SYSTEM StopperingModule (* Module Stoppering, generated from its module specification *)
  (* Standard: 61499-2 *)
  APPLICATION Stoppering (* Module Stoppering on target pc (localhost, IO modbus; generated by modgen) *)
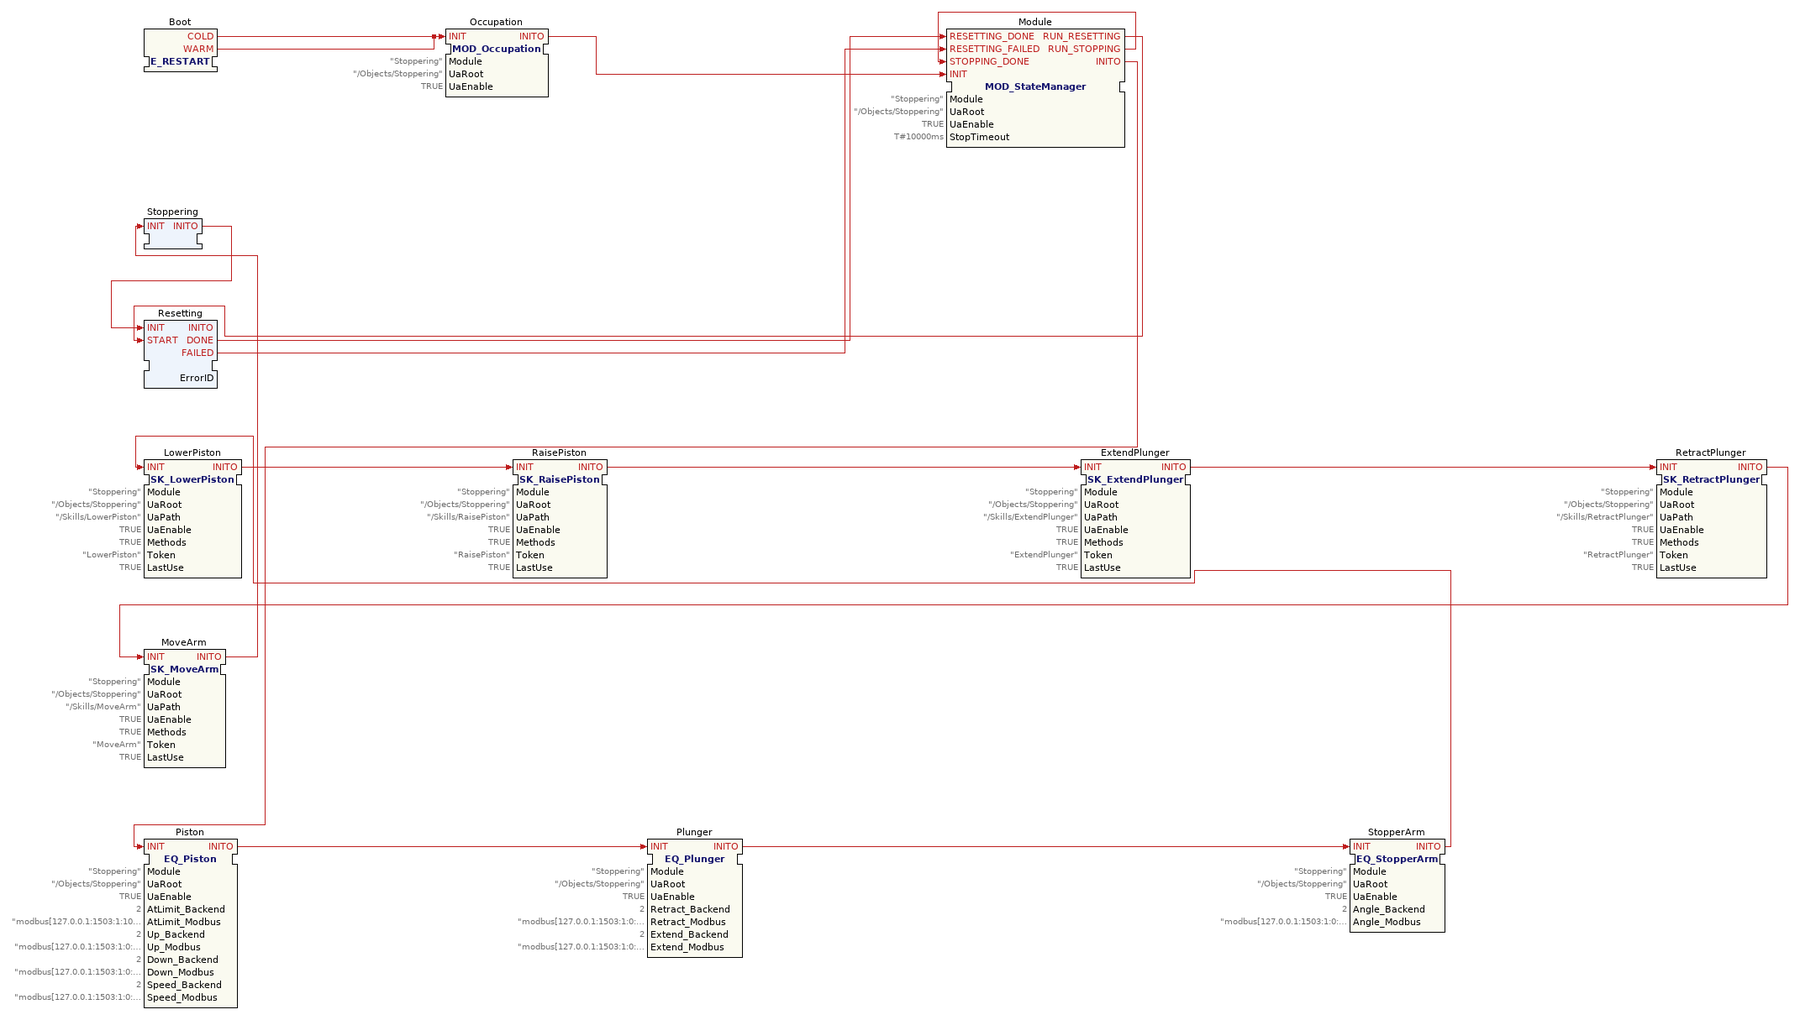
    (* Group ModuleLevel: Module level: occupation, PackML state manager, start-up and the target's IO lines *)
    (* Group ModuleLevelSkills: Module level skills: Control + Execute (+ Stop) sequences of skill primitives; OPC UA /Skills/<name> *)
    (* Group Procedures: Procedures the module state manager runs while Resetting and Stopping *)
    (* Group SkillPrimitives: Skill primitives: one equipment command until a sensor or a time; OPC UA /Skills/<name> *)
    (* Group EquipmentIO: Equipment IO: the only owners of the IO points; skills command them over local channels *)
    FBS
      Boot : iec61499::events::E_RESTART; {SET_ATTRIBUTE(GroupName, ModuleLevel)}
      Occupation : modlib::MOD_Occupation(Module := "Stoppering", UaRoot := "/Objects/Stoppering", UaEnable := TRUE); {SET_ATTRIBUTE(GroupName, ModuleLevel)}
      Module : modlib::MOD_StateManager(Module := "Stoppering", UaRoot := "/Objects/Stoppering", UaEnable := TRUE, StopTimeout := T#10000ms); {SET_ATTRIBUTE(GroupName, ModuleLevel)}
      Piston : stoppering::EQ_Piston(Module := "Stoppering", UaRoot := "/Objects/Stoppering", UaEnable := TRUE, AtLimit_Backend := 2, AtLimit_Modbus := "modbus[127.0.0.1:1503:1:10:d0:]", Up_Backend := 2, Up_Modbus := "modbus[127.0.0.1:1503:1:0::c0]", Down_Backend := 2, Down_Modbus := "modbus[127.0.0.1:1503:1:0::c1]", Speed_Backend := 2, Speed_Modbus := "modbus[127.0.0.1:1503:1:0::h0]"); {SET_ATTRIBUTE(GroupName, EquipmentIO)}
      Plunger : stoppering::EQ_Plunger(Module := "Stoppering", UaRoot := "/Objects/Stoppering", UaEnable := TRUE, Retract_Backend := 2, Retract_Modbus := "modbus[127.0.0.1:1503:1:0::c2]", Extend_Backend := 2, Extend_Modbus := "modbus[127.0.0.1:1503:1:0::c3]"); {SET_ATTRIBUTE(GroupName, EquipmentIO)}
      StopperArm : stoppering::EQ_StopperArm(Module := "Stoppering", UaRoot := "/Objects/Stoppering", UaEnable := TRUE, Angle_Backend := 2, Angle_Modbus := "modbus[127.0.0.1:1503:1:0::h1]"); {SET_ATTRIBUTE(GroupName, EquipmentIO)}
      LowerPiston : stoppering::SK_LowerPiston(Module := "Stoppering", UaRoot := "/Objects/Stoppering", UaPath := "/Skills/LowerPiston", UaEnable := TRUE, Methods := TRUE, Token := "LowerPiston", LastUse := TRUE); {SET_ATTRIBUTE(GroupName, SkillPrimitives)}
      RaisePiston : stoppering::SK_RaisePiston(Module := "Stoppering", UaRoot := "/Objects/Stoppering", UaPath := "/Skills/RaisePiston", UaEnable := TRUE, Methods := TRUE, Token := "RaisePiston", LastUse := TRUE); {SET_ATTRIBUTE(GroupName, SkillPrimitives)}
      ExtendPlunger : stoppering::SK_ExtendPlunger(Module := "Stoppering", UaRoot := "/Objects/Stoppering", UaPath := "/Skills/ExtendPlunger", UaEnable := TRUE, Methods := TRUE, Token := "ExtendPlunger", LastUse := TRUE); {SET_ATTRIBUTE(GroupName, SkillPrimitives)}
      RetractPlunger : stoppering::SK_RetractPlunger(Module := "Stoppering", UaRoot := "/Objects/Stoppering", UaPath := "/Skills/RetractPlunger", UaEnable := TRUE, Methods := TRUE, Token := "RetractPlunger", LastUse := TRUE); {SET_ATTRIBUTE(GroupName, SkillPrimitives)}
      MoveArm : stoppering::SK_MoveArm(Module := "Stoppering", UaRoot := "/Objects/Stoppering", UaPath := "/Skills/MoveArm", UaEnable := TRUE, Methods := TRUE, Token := "MoveArm", LastUse := TRUE); {SET_ATTRIBUTE(GroupName, SkillPrimitives)}
    END_FBS
    SUBAPPLICATION Stoppering (* Module level skill Stoppering: Piston to the working position, place the stopper with the servo, plunge, piston up (runStopperingCycle) *)
      {SET_ATTRIBUTE(GroupName, ModuleLevelSkills)}
      EVENT_INPUT
        INIT : EInit;
      END_EVENT
      EVENT_OUTPUT
        INITO : EInit;
      END_EVENT
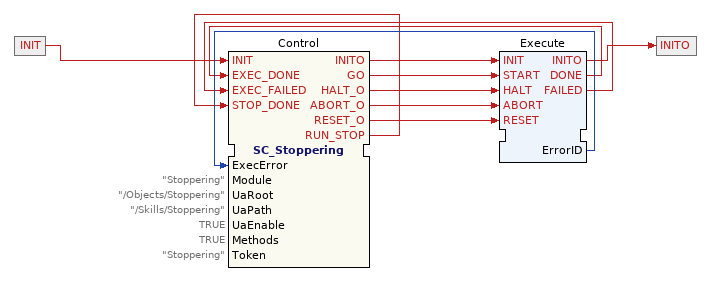
      FBS
        Control : stoppering::SC_Stoppering(Module := "Stoppering", UaRoot := "/Objects/Stoppering", UaPath := "/Skills/Stoppering", UaEnable := TRUE, Methods := TRUE, Token := "Stoppering");
      END_FBS
      SUBAPPLICATION Execute (* Stoppering: execute sequence *)
        EVENT_INPUT
          INIT : EInit;
          START;
          HALT;
          ABORT;
          RESET;
        END_EVENT
        EVENT_OUTPUT
          INITO : EInit;
          DONE;
          FAILED WITH ErrorID;
        END_EVENT
        VAR_OUTPUT
          ErrorID : UINT;
        END_VAR
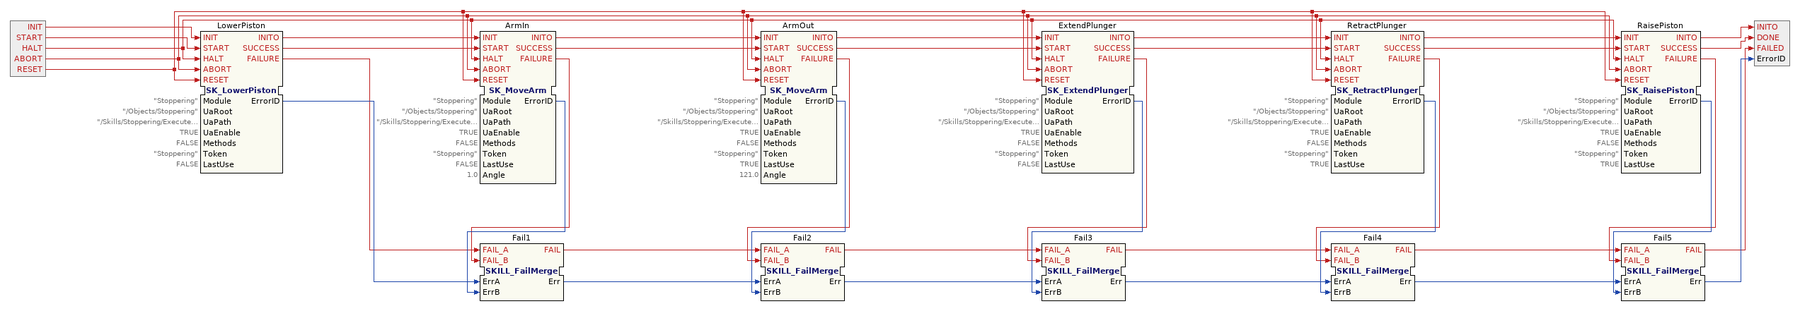
        FBS
          LowerPiston : stoppering::SK_LowerPiston(Module := "Stoppering", UaRoot := "/Objects/Stoppering", UaPath := "/Skills/Stoppering/Execute/LowerPiston", UaEnable := TRUE, Methods := FALSE, Token := "Stoppering", LastUse := FALSE);
          ArmIn : stoppering::SK_MoveArm(Module := "Stoppering", UaRoot := "/Objects/Stoppering", UaPath := "/Skills/Stoppering/Execute/ArmIn", UaEnable := TRUE, Methods := FALSE, Token := "Stoppering", LastUse := FALSE, Angle := 1.0);
          ArmOut : stoppering::SK_MoveArm(Module := "Stoppering", UaRoot := "/Objects/Stoppering", UaPath := "/Skills/Stoppering/Execute/ArmOut", UaEnable := TRUE, Methods := FALSE, Token := "Stoppering", LastUse := TRUE, Angle := 121.0);
          ExtendPlunger : stoppering::SK_ExtendPlunger(Module := "Stoppering", UaRoot := "/Objects/Stoppering", UaPath := "/Skills/Stoppering/Execute/ExtendPlunger", UaEnable := TRUE, Methods := FALSE, Token := "Stoppering", LastUse := FALSE);
          RetractPlunger : stoppering::SK_RetractPlunger(Module := "Stoppering", UaRoot := "/Objects/Stoppering", UaPath := "/Skills/Stoppering/Execute/RetractPlunger", UaEnable := TRUE, Methods := FALSE, Token := "Stoppering", LastUse := TRUE);
          RaisePiston : stoppering::SK_RaisePiston(Module := "Stoppering", UaRoot := "/Objects/Stoppering", UaPath := "/Skills/Stoppering/Execute/RaisePiston", UaEnable := TRUE, Methods := FALSE, Token := "Stoppering", LastUse := TRUE);
          Fail1 : modlib::SKILL_FailMerge;
          Fail2 : modlib::SKILL_FailMerge;
          Fail3 : modlib::SKILL_FailMerge;
          Fail4 : modlib::SKILL_FailMerge;
          Fail5 : modlib::SKILL_FailMerge;
        END_FBS
        EVENT_CONNECTIONS
          INIT TO LowerPiston.INIT;
          RaisePiston.INITO TO INITO;
          START TO LowerPiston.START;
          RaisePiston.SUCCESS TO DONE;
          LowerPiston.INITO TO ArmIn.INIT;
          LowerPiston.SUCCESS TO ArmIn.START;
          ArmIn.INITO TO ArmOut.INIT;
          ArmIn.SUCCESS TO ArmOut.START;
          ArmOut.INITO TO ExtendPlunger.INIT;
          ArmOut.SUCCESS TO ExtendPlunger.START;
          ExtendPlunger.INITO TO RetractPlunger.INIT;
          ExtendPlunger.SUCCESS TO RetractPlunger.START;
          RetractPlunger.INITO TO RaisePiston.INIT;
          RetractPlunger.SUCCESS TO RaisePiston.START;
          HALT TO LowerPiston.HALT;
          HALT TO ArmIn.HALT;
          HALT TO ArmOut.HALT;
          HALT TO ExtendPlunger.HALT;
          HALT TO RetractPlunger.HALT;
          HALT TO RaisePiston.HALT;
          ABORT TO LowerPiston.ABORT;
          ABORT TO ArmIn.ABORT;
          ABORT TO ArmOut.ABORT;
          ABORT TO ExtendPlunger.ABORT;
          ABORT TO RetractPlunger.ABORT;
          ABORT TO RaisePiston.ABORT;
          RESET TO LowerPiston.RESET;
          RESET TO ArmIn.RESET;
          RESET TO ArmOut.RESET;
          RESET TO ExtendPlunger.RESET;
          RESET TO RetractPlunger.RESET;
          RESET TO RaisePiston.RESET;
          LowerPiston.FAILURE TO Fail1.FAIL_A;
          ArmIn.FAILURE TO Fail1.FAIL_B;
          Fail1.FAIL TO Fail2.FAIL_A;
          ArmOut.FAILURE TO Fail2.FAIL_B;
          Fail2.FAIL TO Fail3.FAIL_A;
          ExtendPlunger.FAILURE TO Fail3.FAIL_B;
          Fail3.FAIL TO Fail4.FAIL_A;
          RetractPlunger.FAILURE TO Fail4.FAIL_B;
          Fail4.FAIL TO Fail5.FAIL_A;
          RaisePiston.FAILURE TO Fail5.FAIL_B;
          Fail5.FAIL TO FAILED;
        END_CONNECTIONS
        DATA_CONNECTIONS
          LowerPiston.ErrorID TO Fail1.ErrA;
          ArmIn.ErrorID TO Fail1.ErrB;
          Fail1.Err TO Fail2.ErrA;
          ArmOut.ErrorID TO Fail2.ErrB;
          Fail2.Err TO Fail3.ErrA;
          ExtendPlunger.ErrorID TO Fail3.ErrB;
          Fail3.Err TO Fail4.ErrA;
          RetractPlunger.ErrorID TO Fail4.ErrB;
          Fail4.Err TO Fail5.ErrA;
          RaisePiston.ErrorID TO Fail5.ErrB;
          Fail5.Err TO ErrorID;
        END_CONNECTIONS
      END_SUBAPPLICATION
      EVENT_CONNECTIONS
        INIT TO Control.INIT;
        Control.INITO TO Execute.INIT;
        Control.GO TO Execute.START;
        Control.HALT_O TO Execute.HALT;
        Control.ABORT_O TO Execute.ABORT;
        Control.RESET_O TO Execute.RESET;
        Execute.DONE TO Control.EXEC_DONE;
        Execute.FAILED TO Control.EXEC_FAILED;
        Execute.INITO TO INITO;
        Control.RUN_STOP TO Control.STOP_DONE;
      END_CONNECTIONS
      DATA_CONNECTIONS
        Execute.ErrorID TO Control.ExecError;
      END_CONNECTIONS
    END_SUBAPPLICATION
    SUBAPPLICATION Resetting (* Procedure the module runs while Resetting *)
      {SET_ATTRIBUTE(GroupName, Procedures)}
      EVENT_INPUT
        INIT : EInit;
        START;
      END_EVENT
      EVENT_OUTPUT
        INITO : EInit;
        DONE;
        FAILED WITH ErrorID;
      END_EVENT
      VAR_OUTPUT
        ErrorID : UINT;
      END_VAR
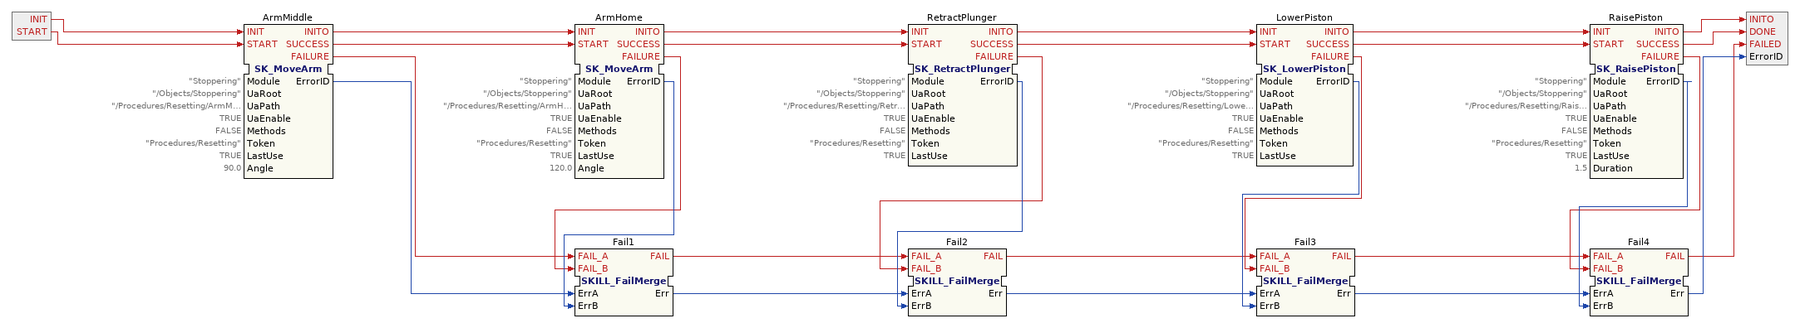
      FBS
        ArmMiddle : stoppering::SK_MoveArm(Module := "Stoppering", UaRoot := "/Objects/Stoppering", UaPath := "/Procedures/Resetting/ArmMiddle", UaEnable := TRUE, Methods := FALSE, Token := "Procedures/Resetting", LastUse := TRUE, Angle := 90.0);
        ArmHome : stoppering::SK_MoveArm(Module := "Stoppering", UaRoot := "/Objects/Stoppering", UaPath := "/Procedures/Resetting/ArmHome", UaEnable := TRUE, Methods := FALSE, Token := "Procedures/Resetting", LastUse := TRUE, Angle := 120.0);
        RetractPlunger : stoppering::SK_RetractPlunger(Module := "Stoppering", UaRoot := "/Objects/Stoppering", UaPath := "/Procedures/Resetting/RetractPlunger", UaEnable := TRUE, Methods := FALSE, Token := "Procedures/Resetting", LastUse := TRUE);
        LowerPiston : stoppering::SK_LowerPiston(Module := "Stoppering", UaRoot := "/Objects/Stoppering", UaPath := "/Procedures/Resetting/LowerPiston", UaEnable := TRUE, Methods := FALSE, Token := "Procedures/Resetting", LastUse := TRUE);
        RaisePiston : stoppering::SK_RaisePiston(Module := "Stoppering", UaRoot := "/Objects/Stoppering", UaPath := "/Procedures/Resetting/RaisePiston", UaEnable := TRUE, Methods := FALSE, Token := "Procedures/Resetting", LastUse := TRUE, Duration := 1.5);
        Fail1 : modlib::SKILL_FailMerge;
        Fail2 : modlib::SKILL_FailMerge;
        Fail3 : modlib::SKILL_FailMerge;
        Fail4 : modlib::SKILL_FailMerge;
      END_FBS
      EVENT_CONNECTIONS
        INIT TO ArmMiddle.INIT;
        RaisePiston.INITO TO INITO;
        START TO ArmMiddle.START;
        RaisePiston.SUCCESS TO DONE;
        ArmMiddle.INITO TO ArmHome.INIT;
        ArmMiddle.SUCCESS TO ArmHome.START;
        ArmHome.INITO TO RetractPlunger.INIT;
        ArmHome.SUCCESS TO RetractPlunger.START;
        RetractPlunger.INITO TO LowerPiston.INIT;
        RetractPlunger.SUCCESS TO LowerPiston.START;
        LowerPiston.INITO TO RaisePiston.INIT;
        LowerPiston.SUCCESS TO RaisePiston.START;
        ArmMiddle.FAILURE TO Fail1.FAIL_A;
        ArmHome.FAILURE TO Fail1.FAIL_B;
        Fail1.FAIL TO Fail2.FAIL_A;
        RetractPlunger.FAILURE TO Fail2.FAIL_B;
        Fail2.FAIL TO Fail3.FAIL_A;
        LowerPiston.FAILURE TO Fail3.FAIL_B;
        Fail3.FAIL TO Fail4.FAIL_A;
        RaisePiston.FAILURE TO Fail4.FAIL_B;
        Fail4.FAIL TO FAILED;
      END_CONNECTIONS
      DATA_CONNECTIONS
        ArmMiddle.ErrorID TO Fail1.ErrA;
        ArmHome.ErrorID TO Fail1.ErrB;
        Fail1.Err TO Fail2.ErrA;
        RetractPlunger.ErrorID TO Fail2.ErrB;
        Fail2.Err TO Fail3.ErrA;
        LowerPiston.ErrorID TO Fail3.ErrB;
        Fail3.Err TO Fail4.ErrA;
        RaisePiston.ErrorID TO Fail4.ErrB;
        Fail4.Err TO ErrorID;
      END_CONNECTIONS
    END_SUBAPPLICATION
    EVENT_CONNECTIONS
      Boot.COLD TO Occupation.INIT;
      Boot.WARM TO Occupation.INIT;
      Module.RUN_RESETTING TO Resetting.START;
      Resetting.DONE TO Module.RESETTING_DONE;
      Resetting.FAILED TO Module.RESETTING_FAILED;
      Module.RUN_STOPPING TO Module.STOPPING_DONE;
      Occupation.INITO TO Module.INIT;
      Module.INITO TO Piston.INIT;
      Piston.INITO TO Plunger.INIT;
      Plunger.INITO TO StopperArm.INIT;
      StopperArm.INITO TO LowerPiston.INIT;
      LowerPiston.INITO TO RaisePiston.INIT;
      RaisePiston.INITO TO ExtendPlunger.INIT;
      ExtendPlunger.INITO TO RetractPlunger.INIT;
      RetractPlunger.INITO TO MoveArm.INIT;
      MoveArm.INITO TO Stoppering.INIT;
      Stoppering.INITO TO Resetting.INIT;
    END_CONNECTIONS
  END_APPLICATION
  APPLICATION Stoppering_pi (* Module Stoppering on target pi (stoppering-pi, IO gpio; generated by modgen) *)
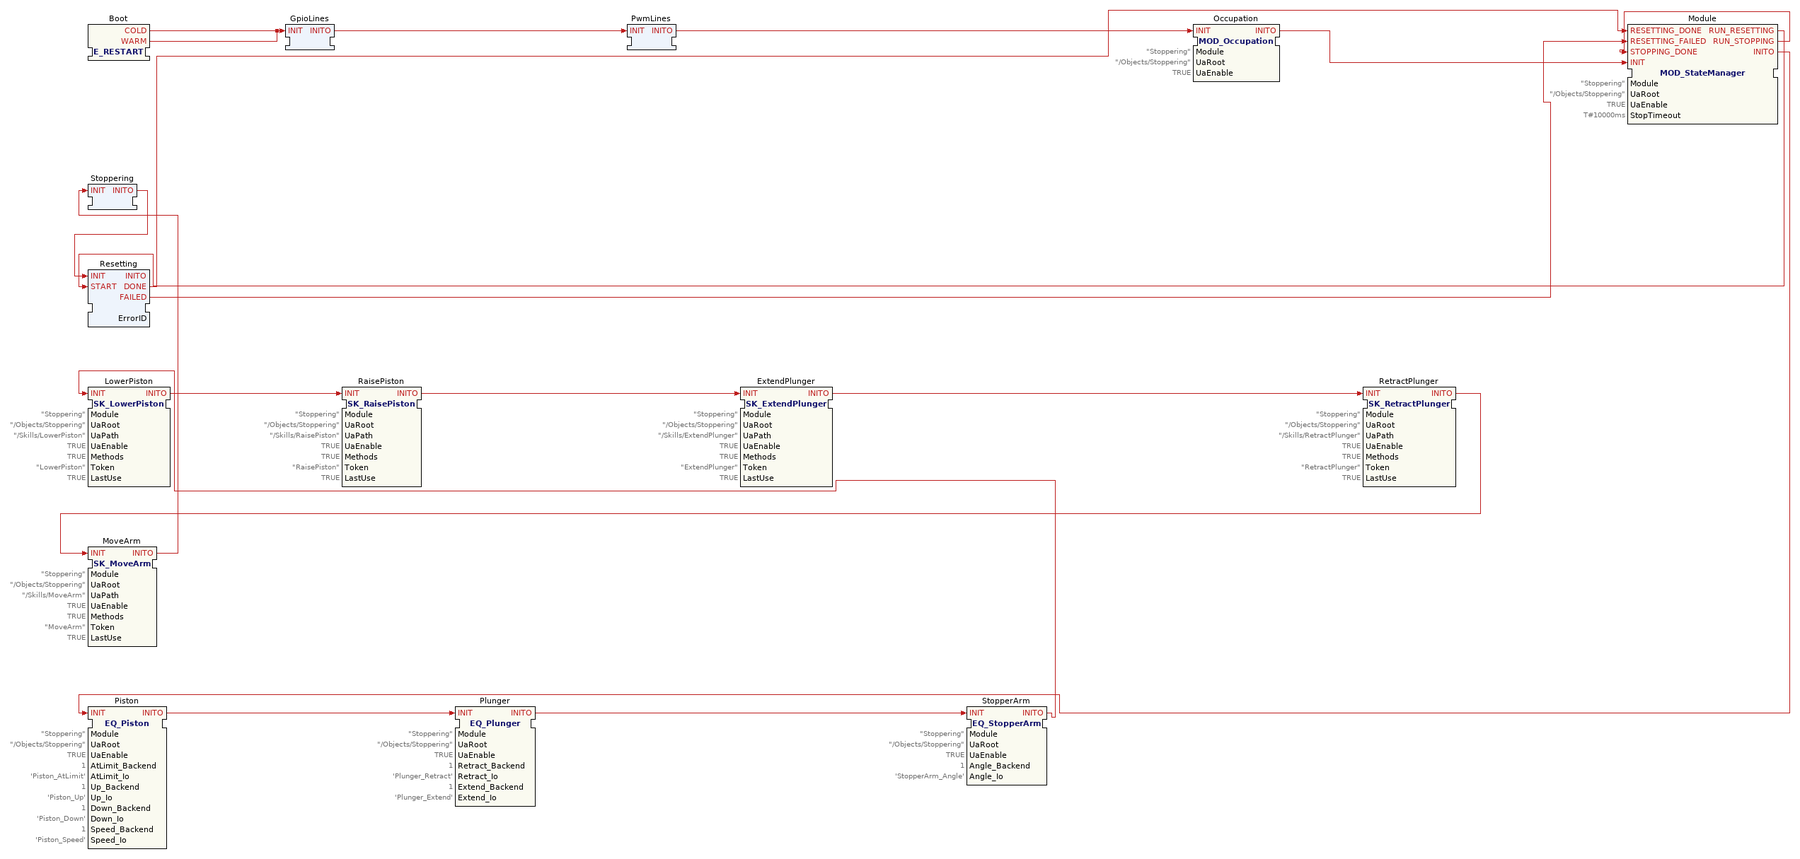
    (* Group ModuleLevel: Module level: occupation, PackML state manager, start-up and the target's IO lines *)
    (* Group ModuleLevelSkills: Module level skills: Control + Execute (+ Stop) sequences of skill primitives; OPC UA /Skills/<name> *)
    (* Group Procedures: Procedures the module state manager runs while Resetting and Stopping *)
    (* Group SkillPrimitives: Skill primitives: one equipment command until a sensor or a time; OPC UA /Skills/<name> *)
    (* Group EquipmentIO: Equipment IO: the only owners of the IO points; skills command them over local channels *)
    FBS
      Boot : iec61499::events::E_RESTART; {SET_ATTRIBUTE(GroupName, ModuleLevel)}
      Occupation : modlib::MOD_Occupation(Module := "Stoppering", UaRoot := "/Objects/Stoppering", UaEnable := TRUE); {SET_ATTRIBUTE(GroupName, ModuleLevel)}
      Module : modlib::MOD_StateManager(Module := "Stoppering", UaRoot := "/Objects/Stoppering", UaEnable := TRUE, StopTimeout := T#10000ms); {SET_ATTRIBUTE(GroupName, ModuleLevel)}
      Piston : stoppering::EQ_Piston(Module := "Stoppering", UaRoot := "/Objects/Stoppering", UaEnable := TRUE, AtLimit_Backend := 1, AtLimit_Io := 'Piston_AtLimit', Up_Backend := 1, Up_Io := 'Piston_Up', Down_Backend := 1, Down_Io := 'Piston_Down', Speed_Backend := 1, Speed_Io := 'Piston_Speed'); {SET_ATTRIBUTE(GroupName, EquipmentIO)}
      Plunger : stoppering::EQ_Plunger(Module := "Stoppering", UaRoot := "/Objects/Stoppering", UaEnable := TRUE, Retract_Backend := 1, Retract_Io := 'Plunger_Retract', Extend_Backend := 1, Extend_Io := 'Plunger_Extend'); {SET_ATTRIBUTE(GroupName, EquipmentIO)}
      StopperArm : stoppering::EQ_StopperArm(Module := "Stoppering", UaRoot := "/Objects/Stoppering", UaEnable := TRUE, Angle_Backend := 1, Angle_Io := 'StopperArm_Angle'); {SET_ATTRIBUTE(GroupName, EquipmentIO)}
      LowerPiston : stoppering::SK_LowerPiston(Module := "Stoppering", UaRoot := "/Objects/Stoppering", UaPath := "/Skills/LowerPiston", UaEnable := TRUE, Methods := TRUE, Token := "LowerPiston", LastUse := TRUE); {SET_ATTRIBUTE(GroupName, SkillPrimitives)}
      RaisePiston : stoppering::SK_RaisePiston(Module := "Stoppering", UaRoot := "/Objects/Stoppering", UaPath := "/Skills/RaisePiston", UaEnable := TRUE, Methods := TRUE, Token := "RaisePiston", LastUse := TRUE); {SET_ATTRIBUTE(GroupName, SkillPrimitives)}
      ExtendPlunger : stoppering::SK_ExtendPlunger(Module := "Stoppering", UaRoot := "/Objects/Stoppering", UaPath := "/Skills/ExtendPlunger", UaEnable := TRUE, Methods := TRUE, Token := "ExtendPlunger", LastUse := TRUE); {SET_ATTRIBUTE(GroupName, SkillPrimitives)}
      RetractPlunger : stoppering::SK_RetractPlunger(Module := "Stoppering", UaRoot := "/Objects/Stoppering", UaPath := "/Skills/RetractPlunger", UaEnable := TRUE, Methods := TRUE, Token := "RetractPlunger", LastUse := TRUE); {SET_ATTRIBUTE(GroupName, SkillPrimitives)}
      MoveArm : stoppering::SK_MoveArm(Module := "Stoppering", UaRoot := "/Objects/Stoppering", UaPath := "/Skills/MoveArm", UaEnable := TRUE, Methods := TRUE, Token := "MoveArm", LastUse := TRUE); {SET_ATTRIBUTE(GroupName, SkillPrimitives)}
    END_FBS
    SUBAPPLICATION GpioLines (* GPIO lines of the equipment's IO points (Linux /dev/gpiochip) *)
      {SET_ATTRIBUTE(GroupName, ModuleLevel)}
      EVENT_INPUT
        INIT : EInit;
      END_EVENT
      EVENT_OUTPUT
        INITO : EInit;
      END_EVENT
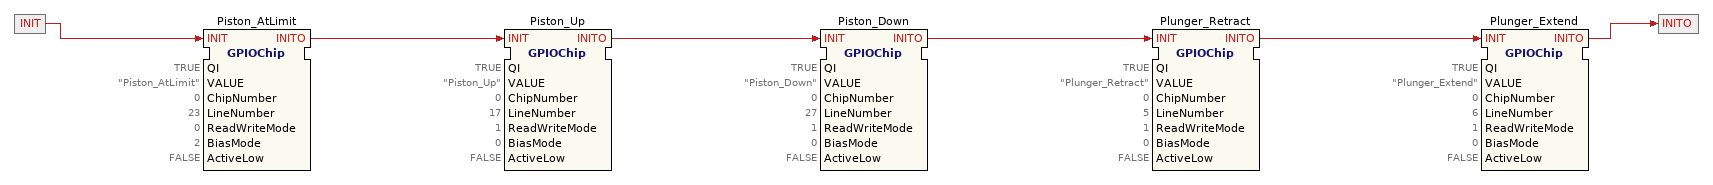
      FBS
        Piston_AtLimit : eclipse4diac::io::gpiochip::GPIOChip(QI := TRUE, VALUE := "Piston_AtLimit", ChipNumber := 0, LineNumber := 23, ReadWriteMode := 0, BiasMode := 2, ActiveLow := FALSE);
        Piston_Up : eclipse4diac::io::gpiochip::GPIOChip(QI := TRUE, VALUE := "Piston_Up", ChipNumber := 0, LineNumber := 17, ReadWriteMode := 1, BiasMode := 0, ActiveLow := FALSE);
        Piston_Down : eclipse4diac::io::gpiochip::GPIOChip(QI := TRUE, VALUE := "Piston_Down", ChipNumber := 0, LineNumber := 27, ReadWriteMode := 1, BiasMode := 0, ActiveLow := FALSE);
        Plunger_Retract : eclipse4diac::io::gpiochip::GPIOChip(QI := TRUE, VALUE := "Plunger_Retract", ChipNumber := 0, LineNumber := 5, ReadWriteMode := 1, BiasMode := 0, ActiveLow := FALSE);
        Plunger_Extend : eclipse4diac::io::gpiochip::GPIOChip(QI := TRUE, VALUE := "Plunger_Extend", ChipNumber := 0, LineNumber := 6, ReadWriteMode := 1, BiasMode := 0, ActiveLow := FALSE);
      END_FBS
      EVENT_CONNECTIONS
        INIT TO Piston_AtLimit.INIT;
        Plunger_Extend.INITO TO INITO;
        Piston_AtLimit.INITO TO Piston_Up.INIT;
        Piston_Up.INITO TO Piston_Down.INIT;
        Piston_Down.INITO TO Plunger_Retract.INIT;
        Plunger_Retract.INITO TO Plunger_Extend.INIT;
      END_CONNECTIONS
    END_SUBAPPLICATION
    SUBAPPLICATION PwmLines (* PWM channels of the equipment's analog outputs (Linux /sys/class/pwm) *)
      {SET_ATTRIBUTE(GroupName, ModuleLevel)}
      EVENT_INPUT
        INIT : EInit;
      END_EVENT
      EVENT_OUTPUT
        INITO : EInit;
      END_EVENT
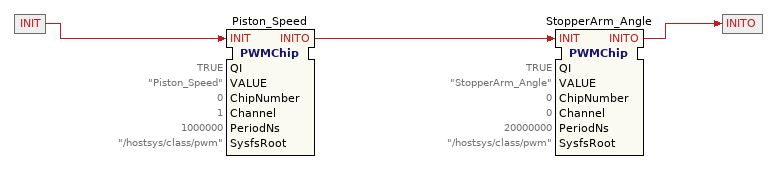
      FBS
        Piston_Speed : eclipse4diac::io::pwmsysfs::PWMChip(QI := TRUE, VALUE := "Piston_Speed", ChipNumber := 0, Channel := 1, PeriodNs := 1000000, SysfsRoot := "/hostsys/class/pwm");
        StopperArm_Angle : eclipse4diac::io::pwmsysfs::PWMChip(QI := TRUE, VALUE := "StopperArm_Angle", ChipNumber := 0, Channel := 0, PeriodNs := 20000000, SysfsRoot := "/hostsys/class/pwm");
      END_FBS
      EVENT_CONNECTIONS
        INIT TO Piston_Speed.INIT;
        StopperArm_Angle.INITO TO INITO;
        Piston_Speed.INITO TO StopperArm_Angle.INIT;
      END_CONNECTIONS
    END_SUBAPPLICATION
    SUBAPPLICATION Stoppering (* Module level skill Stoppering: Piston to the working position, place the stopper with the servo, plunge, piston up (runStopperingCycle) *)
      {SET_ATTRIBUTE(GroupName, ModuleLevelSkills)}
      EVENT_INPUT
        INIT : EInit;
      END_EVENT
      EVENT_OUTPUT
        INITO : EInit;
      END_EVENT
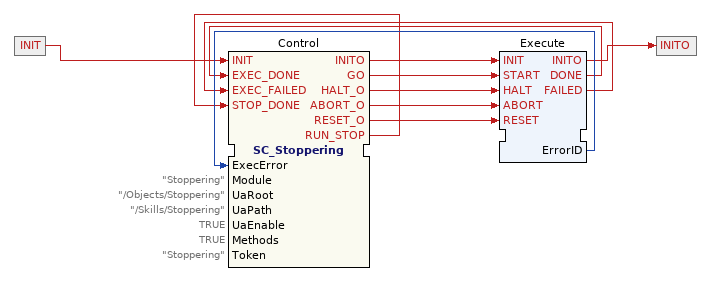
      FBS
        Control : stoppering::SC_Stoppering(Module := "Stoppering", UaRoot := "/Objects/Stoppering", UaPath := "/Skills/Stoppering", UaEnable := TRUE, Methods := TRUE, Token := "Stoppering");
      END_FBS
      SUBAPPLICATION Execute (* Stoppering: execute sequence *)
        EVENT_INPUT
          INIT : EInit;
          START;
          HALT;
          ABORT;
          RESET;
        END_EVENT
        EVENT_OUTPUT
          INITO : EInit;
          DONE;
          FAILED WITH ErrorID;
        END_EVENT
        VAR_OUTPUT
          ErrorID : UINT;
        END_VAR
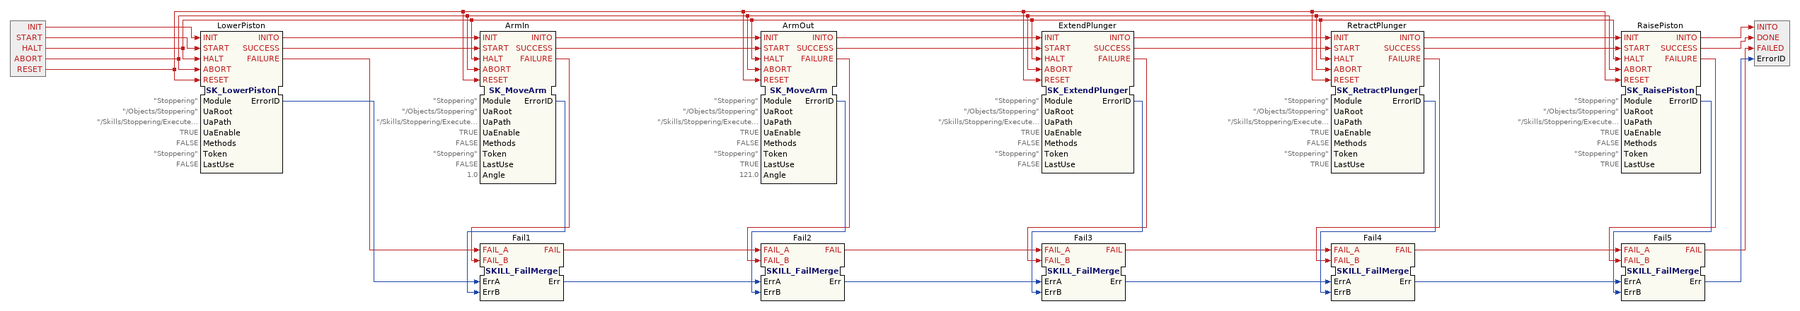
        FBS
          LowerPiston : stoppering::SK_LowerPiston(Module := "Stoppering", UaRoot := "/Objects/Stoppering", UaPath := "/Skills/Stoppering/Execute/LowerPiston", UaEnable := TRUE, Methods := FALSE, Token := "Stoppering", LastUse := FALSE);
          ArmIn : stoppering::SK_MoveArm(Module := "Stoppering", UaRoot := "/Objects/Stoppering", UaPath := "/Skills/Stoppering/Execute/ArmIn", UaEnable := TRUE, Methods := FALSE, Token := "Stoppering", LastUse := FALSE, Angle := 1.0);
          ArmOut : stoppering::SK_MoveArm(Module := "Stoppering", UaRoot := "/Objects/Stoppering", UaPath := "/Skills/Stoppering/Execute/ArmOut", UaEnable := TRUE, Methods := FALSE, Token := "Stoppering", LastUse := TRUE, Angle := 121.0);
          ExtendPlunger : stoppering::SK_ExtendPlunger(Module := "Stoppering", UaRoot := "/Objects/Stoppering", UaPath := "/Skills/Stoppering/Execute/ExtendPlunger", UaEnable := TRUE, Methods := FALSE, Token := "Stoppering", LastUse := FALSE);
          RetractPlunger : stoppering::SK_RetractPlunger(Module := "Stoppering", UaRoot := "/Objects/Stoppering", UaPath := "/Skills/Stoppering/Execute/RetractPlunger", UaEnable := TRUE, Methods := FALSE, Token := "Stoppering", LastUse := TRUE);
          RaisePiston : stoppering::SK_RaisePiston(Module := "Stoppering", UaRoot := "/Objects/Stoppering", UaPath := "/Skills/Stoppering/Execute/RaisePiston", UaEnable := TRUE, Methods := FALSE, Token := "Stoppering", LastUse := TRUE);
          Fail1 : modlib::SKILL_FailMerge;
          Fail2 : modlib::SKILL_FailMerge;
          Fail3 : modlib::SKILL_FailMerge;
          Fail4 : modlib::SKILL_FailMerge;
          Fail5 : modlib::SKILL_FailMerge;
        END_FBS
        EVENT_CONNECTIONS
          INIT TO LowerPiston.INIT;
          RaisePiston.INITO TO INITO;
          START TO LowerPiston.START;
          RaisePiston.SUCCESS TO DONE;
          LowerPiston.INITO TO ArmIn.INIT;
          LowerPiston.SUCCESS TO ArmIn.START;
          ArmIn.INITO TO ArmOut.INIT;
          ArmIn.SUCCESS TO ArmOut.START;
          ArmOut.INITO TO ExtendPlunger.INIT;
          ArmOut.SUCCESS TO ExtendPlunger.START;
          ExtendPlunger.INITO TO RetractPlunger.INIT;
          ExtendPlunger.SUCCESS TO RetractPlunger.START;
          RetractPlunger.INITO TO RaisePiston.INIT;
          RetractPlunger.SUCCESS TO RaisePiston.START;
          HALT TO LowerPiston.HALT;
          HALT TO ArmIn.HALT;
          HALT TO ArmOut.HALT;
          HALT TO ExtendPlunger.HALT;
          HALT TO RetractPlunger.HALT;
          HALT TO RaisePiston.HALT;
          ABORT TO LowerPiston.ABORT;
          ABORT TO ArmIn.ABORT;
          ABORT TO ArmOut.ABORT;
          ABORT TO ExtendPlunger.ABORT;
          ABORT TO RetractPlunger.ABORT;
          ABORT TO RaisePiston.ABORT;
          RESET TO LowerPiston.RESET;
          RESET TO ArmIn.RESET;
          RESET TO ArmOut.RESET;
          RESET TO ExtendPlunger.RESET;
          RESET TO RetractPlunger.RESET;
          RESET TO RaisePiston.RESET;
          LowerPiston.FAILURE TO Fail1.FAIL_A;
          ArmIn.FAILURE TO Fail1.FAIL_B;
          Fail1.FAIL TO Fail2.FAIL_A;
          ArmOut.FAILURE TO Fail2.FAIL_B;
          Fail2.FAIL TO Fail3.FAIL_A;
          ExtendPlunger.FAILURE TO Fail3.FAIL_B;
          Fail3.FAIL TO Fail4.FAIL_A;
          RetractPlunger.FAILURE TO Fail4.FAIL_B;
          Fail4.FAIL TO Fail5.FAIL_A;
          RaisePiston.FAILURE TO Fail5.FAIL_B;
          Fail5.FAIL TO FAILED;
        END_CONNECTIONS
        DATA_CONNECTIONS
          LowerPiston.ErrorID TO Fail1.ErrA;
          ArmIn.ErrorID TO Fail1.ErrB;
          Fail1.Err TO Fail2.ErrA;
          ArmOut.ErrorID TO Fail2.ErrB;
          Fail2.Err TO Fail3.ErrA;
          ExtendPlunger.ErrorID TO Fail3.ErrB;
          Fail3.Err TO Fail4.ErrA;
          RetractPlunger.ErrorID TO Fail4.ErrB;
          Fail4.Err TO Fail5.ErrA;
          RaisePiston.ErrorID TO Fail5.ErrB;
          Fail5.Err TO ErrorID;
        END_CONNECTIONS
      END_SUBAPPLICATION
      EVENT_CONNECTIONS
        INIT TO Control.INIT;
        Control.INITO TO Execute.INIT;
        Control.GO TO Execute.START;
        Control.HALT_O TO Execute.HALT;
        Control.ABORT_O TO Execute.ABORT;
        Control.RESET_O TO Execute.RESET;
        Execute.DONE TO Control.EXEC_DONE;
        Execute.FAILED TO Control.EXEC_FAILED;
        Execute.INITO TO INITO;
        Control.RUN_STOP TO Control.STOP_DONE;
      END_CONNECTIONS
      DATA_CONNECTIONS
        Execute.ErrorID TO Control.ExecError;
      END_CONNECTIONS
    END_SUBAPPLICATION
    SUBAPPLICATION Resetting (* Procedure the module runs while Resetting *)
      {SET_ATTRIBUTE(GroupName, Procedures)}
      EVENT_INPUT
        INIT : EInit;
        START;
      END_EVENT
      EVENT_OUTPUT
        INITO : EInit;
        DONE;
        FAILED WITH ErrorID;
      END_EVENT
      VAR_OUTPUT
        ErrorID : UINT;
      END_VAR
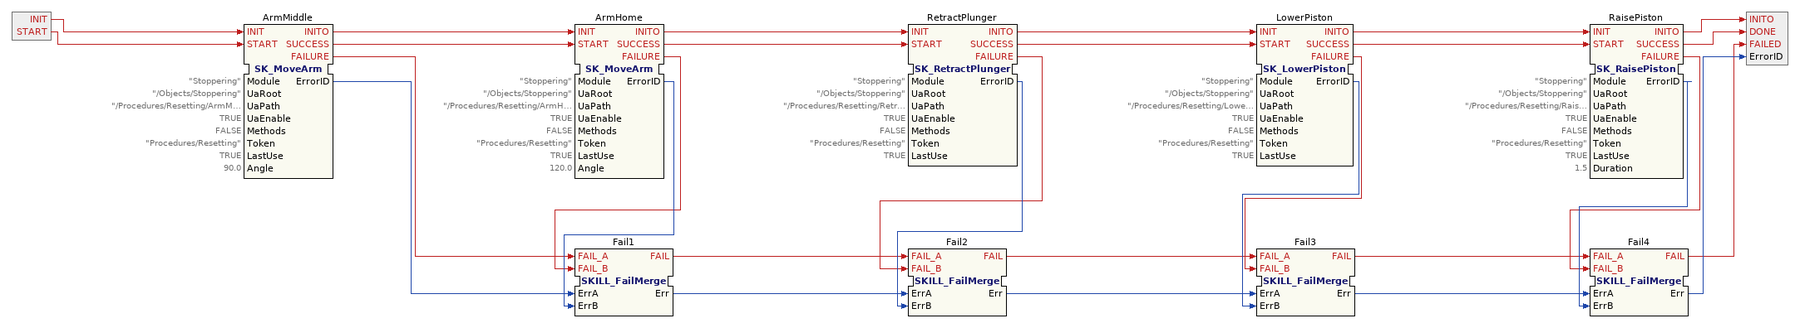
      FBS
        ArmMiddle : stoppering::SK_MoveArm(Module := "Stoppering", UaRoot := "/Objects/Stoppering", UaPath := "/Procedures/Resetting/ArmMiddle", UaEnable := TRUE, Methods := FALSE, Token := "Procedures/Resetting", LastUse := TRUE, Angle := 90.0);
        ArmHome : stoppering::SK_MoveArm(Module := "Stoppering", UaRoot := "/Objects/Stoppering", UaPath := "/Procedures/Resetting/ArmHome", UaEnable := TRUE, Methods := FALSE, Token := "Procedures/Resetting", LastUse := TRUE, Angle := 120.0);
        RetractPlunger : stoppering::SK_RetractPlunger(Module := "Stoppering", UaRoot := "/Objects/Stoppering", UaPath := "/Procedures/Resetting/RetractPlunger", UaEnable := TRUE, Methods := FALSE, Token := "Procedures/Resetting", LastUse := TRUE);
        LowerPiston : stoppering::SK_LowerPiston(Module := "Stoppering", UaRoot := "/Objects/Stoppering", UaPath := "/Procedures/Resetting/LowerPiston", UaEnable := TRUE, Methods := FALSE, Token := "Procedures/Resetting", LastUse := TRUE);
        RaisePiston : stoppering::SK_RaisePiston(Module := "Stoppering", UaRoot := "/Objects/Stoppering", UaPath := "/Procedures/Resetting/RaisePiston", UaEnable := TRUE, Methods := FALSE, Token := "Procedures/Resetting", LastUse := TRUE, Duration := 1.5);
        Fail1 : modlib::SKILL_FailMerge;
        Fail2 : modlib::SKILL_FailMerge;
        Fail3 : modlib::SKILL_FailMerge;
        Fail4 : modlib::SKILL_FailMerge;
      END_FBS
      EVENT_CONNECTIONS
        INIT TO ArmMiddle.INIT;
        RaisePiston.INITO TO INITO;
        START TO ArmMiddle.START;
        RaisePiston.SUCCESS TO DONE;
        ArmMiddle.INITO TO ArmHome.INIT;
        ArmMiddle.SUCCESS TO ArmHome.START;
        ArmHome.INITO TO RetractPlunger.INIT;
        ArmHome.SUCCESS TO RetractPlunger.START;
        RetractPlunger.INITO TO LowerPiston.INIT;
        RetractPlunger.SUCCESS TO LowerPiston.START;
        LowerPiston.INITO TO RaisePiston.INIT;
        LowerPiston.SUCCESS TO RaisePiston.START;
        ArmMiddle.FAILURE TO Fail1.FAIL_A;
        ArmHome.FAILURE TO Fail1.FAIL_B;
        Fail1.FAIL TO Fail2.FAIL_A;
        RetractPlunger.FAILURE TO Fail2.FAIL_B;
        Fail2.FAIL TO Fail3.FAIL_A;
        LowerPiston.FAILURE TO Fail3.FAIL_B;
        Fail3.FAIL TO Fail4.FAIL_A;
        RaisePiston.FAILURE TO Fail4.FAIL_B;
        Fail4.FAIL TO FAILED;
      END_CONNECTIONS
      DATA_CONNECTIONS
        ArmMiddle.ErrorID TO Fail1.ErrA;
        ArmHome.ErrorID TO Fail1.ErrB;
        Fail1.Err TO Fail2.ErrA;
        RetractPlunger.ErrorID TO Fail2.ErrB;
        Fail2.Err TO Fail3.ErrA;
        LowerPiston.ErrorID TO Fail3.ErrB;
        Fail3.Err TO Fail4.ErrA;
        RaisePiston.ErrorID TO Fail4.ErrB;
        Fail4.Err TO ErrorID;
      END_CONNECTIONS
    END_SUBAPPLICATION
    EVENT_CONNECTIONS
      Boot.COLD TO GpioLines.INIT;
      Boot.WARM TO GpioLines.INIT;
      Module.RUN_RESETTING TO Resetting.START;
      Resetting.DONE TO Module.RESETTING_DONE;
      Resetting.FAILED TO Module.RESETTING_FAILED;
      Module.RUN_STOPPING TO Module.STOPPING_DONE;
      GpioLines.INITO TO PwmLines.INIT;
      PwmLines.INITO TO Occupation.INIT;
      Occupation.INITO TO Module.INIT;
      Module.INITO TO Piston.INIT;
      Piston.INITO TO Plunger.INIT;
      Plunger.INITO TO StopperArm.INIT;
      StopperArm.INITO TO LowerPiston.INIT;
      LowerPiston.INITO TO RaisePiston.INIT;
      RaisePiston.INITO TO ExtendPlunger.INIT;
      ExtendPlunger.INITO TO RetractPlunger.INIT;
      RetractPlunger.INITO TO MoveArm.INIT;
      MoveArm.INITO TO Stoppering.INIT;
      Stoppering.INITO TO Resetting.INIT;
    END_CONNECTIONS
  END_APPLICATION
  DEVICE FORTE_PC : iec61499::system::FORTE_PC(MGR_ID := "localhost:61499")
    {SET_ATTRIBUTE(Profile, HOLOBLOC)} (* device profile *)
    RESOURCE RES : iec61499::system::EMB_RES
    END_RESOURCE
  END_DEVICE
  DEVICE FORTE_PI : iec61499::system::FORTE_PC(MGR_ID := "stoppering-pi:61499")
    {SET_ATTRIBUTE(Profile, HOLOBLOC)} (* device profile *)
    RESOURCE RES : iec61499::system::EMB_RES
    END_RESOURCE
  END_DEVICE
  MAPPINGS
    Stoppering.Boot ON FORTE_PC.RES;
    Stoppering.Occupation ON FORTE_PC.RES;
    Stoppering.Module ON FORTE_PC.RES;
    Stoppering.Piston ON FORTE_PC.RES;
    Stoppering.Plunger ON FORTE_PC.RES;
    Stoppering.StopperArm ON FORTE_PC.RES;
    Stoppering.LowerPiston ON FORTE_PC.RES;
    Stoppering.RaisePiston ON FORTE_PC.RES;
    Stoppering.ExtendPlunger ON FORTE_PC.RES;
    Stoppering.RetractPlunger ON FORTE_PC.RES;
    Stoppering.MoveArm ON FORTE_PC.RES;
    Stoppering.Stoppering ON FORTE_PC.RES;
    Stoppering.Resetting ON FORTE_PC.RES;
    Stoppering_pi.Boot ON FORTE_PI.RES;
    Stoppering_pi.Occupation ON FORTE_PI.RES;
    Stoppering_pi.Module ON FORTE_PI.RES;
    Stoppering_pi.GpioLines ON FORTE_PI.RES;
    Stoppering_pi.PwmLines ON FORTE_PI.RES;
    Stoppering_pi.Piston ON FORTE_PI.RES;
    Stoppering_pi.Plunger ON FORTE_PI.RES;
    Stoppering_pi.StopperArm ON FORTE_PI.RES;
    Stoppering_pi.LowerPiston ON FORTE_PI.RES;
    Stoppering_pi.RaisePiston ON FORTE_PI.RES;
    Stoppering_pi.ExtendPlunger ON FORTE_PI.RES;
    Stoppering_pi.RetractPlunger ON FORTE_PI.RES;
    Stoppering_pi.MoveArm ON FORTE_PI.RES;
    Stoppering_pi.Stoppering ON FORTE_PI.RES;
    Stoppering_pi.Resetting ON FORTE_PI.RES;
  END_MAPPINGS
END_SYSTEM
